% RSLogix 500 project Project1.RSS, saved by version 8.30.00.16 %
PROJECT "PROC1"    % processor: Bul.1763 MicroLogix 1100 Series B %

PROGRAM FILES
  LAD 2 "MAIN"  10 rungs
  LAD 3 "I0"  5 rungs

DATA FILES
  O0 OUTPUT  5 elements
  I1 INPUT  7 elements
  S2 STATUS  66 elements
  B3 BINARY  1 elements
  T4 TIMER  3 elements
  C5 COUNTER  1 elements
  R6 CONTROL  1 elements
  N7 INTEGER  1 elements
  F8 FLOAT  1 elements

LADDER 2 "MAIN"
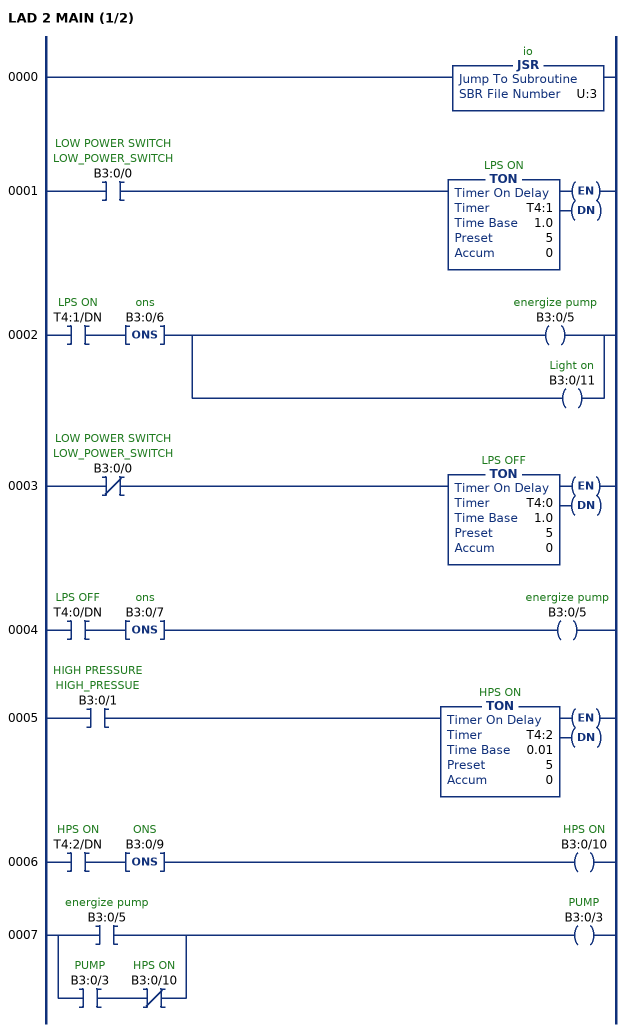
% Rung: 0 %
SOR JSR U:3 EOR
%   U:3  "io" %
% Rung: 1 %
SOR XIC B3:0/0 TON T4:1 1.0 5 0 EOR
%   B3:0/0  LOW_POWER_SWITCH  "LOW POWER SWITCH" %
%   T4:1  "LPS ON" %
% Rung: 2 %
SOR XIC T4:1/DN ONS B3:0/6 BST OTE B3:0/5 NXB OTE B3:0/11 BND EOR
%   T4:1/DN  "LPS ON" %
%   B3:0/6  "ons" %
%   B3:0/5  "energize pump" %
%   B3:0/11  "Light on" %
% Rung: 3 %
SOR XIO B3:0/0 TON T4:0 1.0 5 0 EOR
%   B3:0/0  LOW_POWER_SWITCH  "LOW POWER SWITCH" %
%   T4:0  "LPS OFF" %
% Rung: 4 %
SOR XIC T4:0/DN ONS B3:0/7 OTE B3:0/5 EOR
%   T4:0/DN  "LPS OFF" %
%   B3:0/7  "ons" %
%   B3:0/5  "energize pump" %
% Rung: 5 %
SOR XIC B3:0/1 TON T4:2 0.01 5 0 EOR
%   B3:0/1  HIGH_PRESSUE  "HIGH PRESSURE" %
%   T4:2  "HPS ON" %
% Rung: 6 %
SOR XIC T4:2/DN ONS B3:0/9 OTE B3:0/10 EOR
%   T4:2/DN  "HPS ON" %
%   B3:0/9  "ONS" %
%   B3:0/10  "HPS ON" %
% Rung: 7 %
SOR BST XIC B3:0/5 NXB XIC B3:0/3 XIO B3:0/10 BND OTE B3:0/3 EOR
%   B3:0/5  "energize pump" %
%   B3:0/3  "PUMP" %
%   B3:0/10  "HPS ON" %

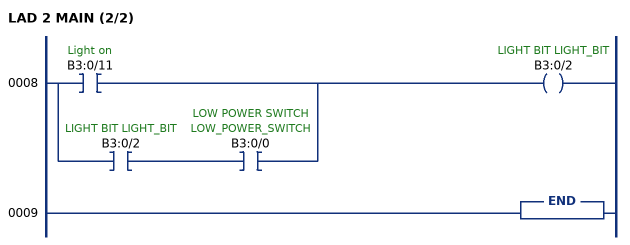
% Rung: 8 %
SOR BST XIC B3:0/11 NXB XIC B3:0/2 XIC B3:0/0 BND OTE B3:0/2 EOR
%   B3:0/11  "Light on" %
%   B3:0/2  LIGHT_BIT  "LIGHT BIT" %
%   B3:0/0  LOW_POWER_SWITCH  "LOW POWER SWITCH" %
% Rung: 9 %
SOR END EOR

LADDER 3 "I0"
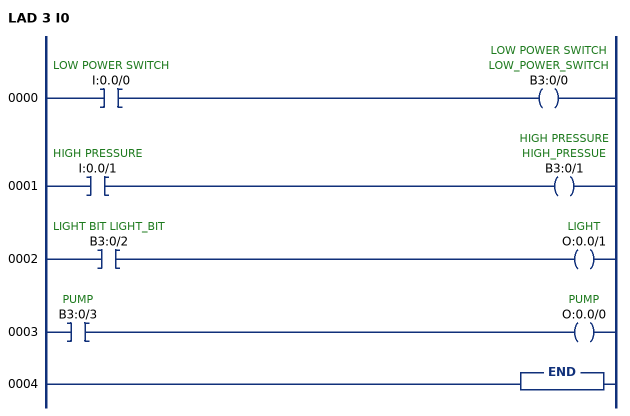
% Rung: 0 %
SOR XIC I:0.0/0 OTE B3:0/0 EOR
%   I:0.0/0  "LOW POWER SWITCH" %
%   B3:0/0  LOW_POWER_SWITCH  "LOW POWER SWITCH" %
% Rung: 1 %
SOR XIC I:0.0/1 OTE B3:0/1 EOR
%   I:0.0/1  "HIGH PRESSURE" %
%   B3:0/1  HIGH_PRESSUE  "HIGH PRESSURE" %
% Rung: 2 %
SOR XIC B3:0/2 OTE O:0.0/1 EOR
%   B3:0/2  LIGHT_BIT  "LIGHT BIT" %
%   O:0.0/1  "LIGHT" %
% Rung: 3 %
SOR XIC B3:0/3 OTE O:0.0/0 EOR
%   B3:0/3  "PUMP" %
%   O:0.0/0  "PUMP" %
% Rung: 4 %
SOR END EOR

OTHER DOCUMENTED ADDRESSES
  B3:0/8  "pump <90"
  B3:5  "energize"
  B3:6  "oneshot"
  I:1.0/0  "PRESSURE SWITCH"
  U:4  "INPUTS"

REVISION NOTES
  0: debugg
  1: debugg
  2: dedugg
  3: FINAL VERSION
  4: FINAL
  5: FINAL
  6: FINAL VERSION
  7: Fina; version
  8: final version
  9: project with timers
  10: With timers
  11: with timers
  12: Final version with timers

DATA TABLE (non-zero values as saved)
DATA T4
% .PRE .ACC %
% T4:0 % 5 0
% T4:1 % 5 0
% T4:2 % 5 0
